// TIA Portal V18 export
// export: Created 2026-03-12T15:56:18.9615037Z, ExportSetting WithDefaults, DisplayName Totally Integrated Automation Portal, DisplayVersion V18 Update 5, DisplayName TIA Portal Openness, DisplayVersion V18 Update 5, DisplayName TIA Portal Version Control Interface, DisplayVersion V18, DisplayName SINAMICS Startdrive Advanced, DisplayVersion V18, DisplayName SINAMICS Startdrive G130, G150, S120, S150, SINAMICS MV, S210, DisplayVersion V18, DisplayName SINAMICS Startdrive G110M, G120, G120C, G120D, G120P, G115D, DisplayVersion V18, DisplayName STEP 7 Professional, DisplayVersion V18 Update 5, DisplayName STEP 7 Safety, DisplayVersion V18, DisplayName WinCC Professional, DisplayVersion V18 Update 5
DATA_BLOCK "FB FALHA BH-01A"   // DB211
VERSION : 0.1
// stored: AutoNumber true, DBAccessibleFromOPCUA true, DBAccessibleFromWebserver true, InstanceOfName FB FALHA, InstanceOfType FB
"FB FALHA"
   // VAR_INPUT
   //    INPUT_FALHA : Bool;
   //    INPUT_TEMPO_RESET : Time;
   //    INPUT_TEMPO_NÃO_LIGOU : Time;
   //    INPUT_LIGADO : Bool;
   //    INPUT_RESET_FALHA : Bool;
   //    INPUT_SAIDA_LIGA_BOMBA : Bool;
   //    INPUT_HABILITA_CONJUNTO : Bool;
   //    INPUT_MANUTENCAO : Bool;
   // END_VAR
   // VAR_OUTPUT
   //    FALHA : Bool;
   //    RESET_FALHA_INVERSOR : Bool;
   //    FALHA_NÃO_LIGOU : Bool;
   // END_VAR
   // VAR
   //    NÃO_LIGOU : Bool;
   //    SET_FALHA : Bool;
   //    TIMER_1 : IEC_TIMER;
   //    TIMER_2 : IEC_TIMER;
   //    LIGA_BOMBA_AUX { S7_SetPoint := 'True'} : Bool;
   // END_VAR
BEGIN
END_DATA_BLOCK
